// TIA Portal V17 export
// export: Created 2024-09-02T12:49:55.5450562Z, ExportSetting WithDefaults, DisplayName Totally Integrated Automation Portal, DisplayVersion V17, DisplayName TIA Portal Openness, DisplayVersion V17, DisplayName TIA Portal Version Control Interface, DisplayVersion V17, DisplayName STEP 7 Professional, DisplayVersion V17, DisplayName STEP 7 Safety, DisplayVersion V17, DisplayName WinCC Professional, DisplayVersion V17
FUNCTION "SysFC_HMI_Functions" : Void   // FC251, LAD
TITLE = Power supply for function lines / Versorgung Funktionszeilen
{ S7_Optimized_Access := 'TRUE' }
AUTHOR : OlegFuehrus
FAMILY : HMI
NAME : HMI
VERSION : 1.0
// stored: AutoNumber true, IsIECCheckEnabled false, SetENOAutomatically false, UDAEnableTagReadback false
   VAR_INPUT
      "Type" : WString;   // Typ (Setup, PowerUp, Unit, NutRunner, NutRunnerGroup, CycleType, UserDefine) / Type (Setup, PowerUp, Unit, NutRunner, NutRunnerGroup, CycleType, UserDefine)
      Line : Int;   // Zeile (1..348) / Line (1. . 348)
      "Enable Left" : Bool;   // Funktionsfreigabe Links / Functional Approve
      "Enable Right" : Bool;   // Funktionsfreigabe Rechts / Function release right
      "End Pos. Left" : Bool;   // Endlage Links (gelb) / End position Left (yellow)
      "End Pos. Right" : Bool;   // Endlage Rechts (gruen) / End position right (green)
      Position : LReal;   // Positionsanzeige / position display
      "Hide Pos." : Bool;   // Position ausblenden / Hide position
      "Hide Left Arrow" : Bool;   // Pfeil Links ausblenden / Hide left arrow
      "Hide Right Arrow" : Bool;   // Pfeil Rechts ausblenden / Hide left arrow
   END_VAR
   VAR_OUTPUT
      Function_left : Bool;   // Funktionstaste links / Function key left
      Function_right : Bool;   // Funktionstaste rechts / Function key right
      ConfigFault : Bool;   // Configurationsfehler / configuration error
   END_VAR
   VAR_IN_OUT
      LTLL_Config : "LTLL_typeConfig";
      LTLL_Data : "LTLL_typeData";
   END_VAR
   VAR_TEMP
      t_RetVal : Word;
      t_VKE0 : Bool;
      t_VKE1 : Bool;
      t_ConfigFault : Bool;
      t_ConfigFaultNr : Int;
      t_Line : Int;
      t_Line_Uint : UInt;
      t_Btn_Left : Bool;
      t_Btn_Right : Bool;
      t_secure_bit_ok : Bool;
      t_ErrID : Word;
      t_loop : Int;
      t_Pointer : Int;
      t_CmpOK : Bool;
      t_PowerUp : Bool;
   END_VAR
BEGIN

REGION Network 1: VKE0
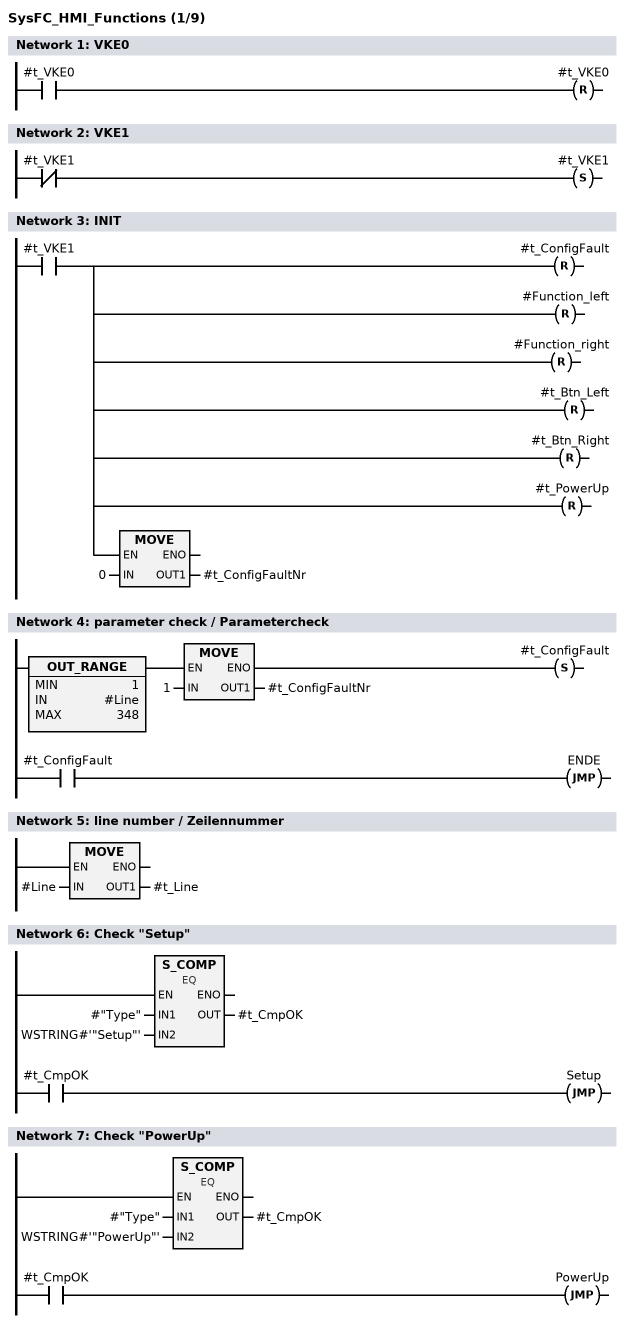
   RUNG wire#powerrail
      Contact( #t_VKE0 )
      R_Coil( #t_VKE0 )
   END_RUNG
   // the same network as SCL:
   IF #t_VKE0 THEN #t_VKE0 := FALSE; END_IF;
END_REGION

REGION Network 2: VKE1
   RUNG wire#powerrail
      I_Contact( #t_VKE1 )
      S_Coil( #t_VKE1 )
   END_RUNG
   // the same network as SCL:
   IF NOT #t_VKE1 THEN #t_VKE1 := TRUE; END_IF;
END_REGION

REGION Network 3: INIT
   RUNG wire#powerrail
      Contact( #t_VKE1 )
      wire#w1
      R_Coil( #t_ConfigFault )
   END_RUNG
   RUNG wire#w1
      R_Coil( #Function_left )
   END_RUNG
   RUNG wire#w1
      R_Coil( #Function_right )
   END_RUNG
   RUNG wire#w1
      R_Coil( #t_Btn_Left )
   END_RUNG
   RUNG wire#w1
      R_Coil( #t_Btn_Right )
   END_RUNG
   RUNG wire#w1
      R_Coil( #t_PowerUp )
   END_RUNG
   RUNG wire#w1
      Move(in := 0, out1 => #t_ConfigFaultNr)
   END_RUNG
   // the same network as SCL:
   IF #t_VKE1 THEN
       #t_ConfigFault := FALSE;
       #Function_left := FALSE;
       #Function_right := FALSE;
       #t_Btn_Left := FALSE;
       #t_Btn_Right := FALSE;
       #t_PowerUp := FALSE;
       #t_ConfigFaultNr := 0;
   END_IF;
END_REGION

REGION Network 4: parameter check / Parametercheck
   IF (#Line < 1) OR (#Line > 348) THEN
       #t_ConfigFaultNr := 1;
       #t_ConfigFault := TRUE;
   END_IF;
   IF #t_ConfigFault THEN GOTO ENDE; END_IF;
END_REGION

REGION Network 5: line number / Zeilennummer
   RUNG wire#powerrail
      Move(in := #Line, out1 => #t_Line)
   END_RUNG
   // the same network as SCL:
   #t_Line := #Line;
END_REGION

REGION Network 6: Check "Setup"
   RUNG wire#powerrail
      { S7_Templates := "[relation := EQ, src_type := WString]" } S_COMP(IN1 := #"Type", IN2 := WSTRING#'"Setup"', OUT => #t_CmpOK)
   END_RUNG
   RUNG wire#powerrail
      Contact( #t_CmpOK )
      JumpCoil( Setup )
   END_RUNG
   // the same network as SCL:
   S_COMP(IN1 := #"Type", IN2 := WSTRING#'"Setup"', OUT => #t_CmpOK);
   IF #t_CmpOK THEN GOTO Setup; END_IF;
END_REGION

REGION Network 7: Check "PowerUp"
   RUNG wire#powerrail
      { S7_Templates := "[relation := EQ, src_type := WString]" } S_COMP(IN1 := #"Type", IN2 := WSTRING#'"PowerUp"', OUT => #t_CmpOK)
   END_RUNG
   RUNG wire#powerrail
      Contact( #t_CmpOK )
      JumpCoil( PowerUp )
   END_RUNG
   // the same network as SCL:
   S_COMP(IN1 := #"Type", IN2 := WSTRING#'"PowerUp"', OUT => #t_CmpOK);
   IF #t_CmpOK THEN GOTO PowerUp; END_IF;
END_REGION

REGION Network 8: Check "Unit"
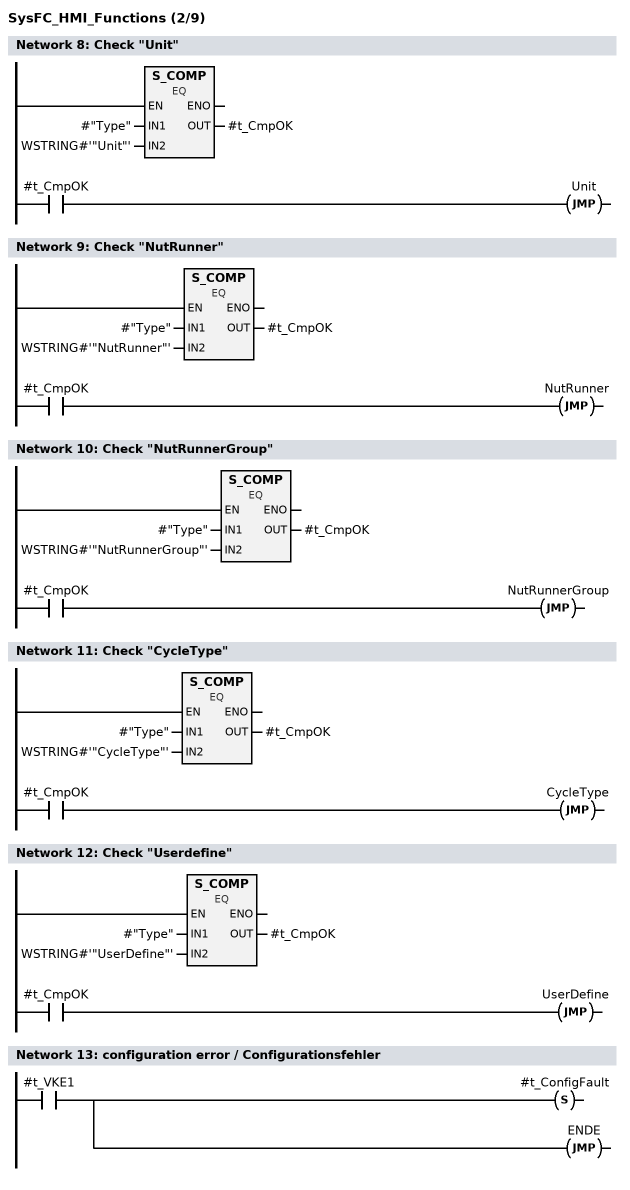
   RUNG wire#powerrail
      { S7_Templates := "[relation := EQ, src_type := WString]" } S_COMP(IN1 := #"Type", IN2 := WSTRING#'"Unit"', OUT => #t_CmpOK)
   END_RUNG
   RUNG wire#powerrail
      Contact( #t_CmpOK )
      JumpCoil( Unit )
   END_RUNG
   // the same network as SCL:
   S_COMP(IN1 := #"Type", IN2 := WSTRING#'"Unit"', OUT => #t_CmpOK);
   IF #t_CmpOK THEN GOTO Unit; END_IF;
END_REGION

REGION Network 9: Check "NutRunner"
   RUNG wire#powerrail
      { S7_Templates := "[relation := EQ, src_type := WString]" } S_COMP(IN1 := #"Type", IN2 := WSTRING#'"NutRunner"', OUT => #t_CmpOK)
   END_RUNG
   RUNG wire#powerrail
      Contact( #t_CmpOK )
      JumpCoil( NutRunner )
   END_RUNG
   // the same network as SCL:
   S_COMP(IN1 := #"Type", IN2 := WSTRING#'"NutRunner"', OUT => #t_CmpOK);
   IF #t_CmpOK THEN GOTO NutRunner; END_IF;
END_REGION

REGION Network 10: Check "NutRunnerGroup"
   RUNG wire#powerrail
      { S7_Templates := "[relation := EQ, src_type := WString]" } S_COMP(IN1 := #"Type", IN2 := WSTRING#'"NutRunnerGroup"', OUT => #t_CmpOK)
   END_RUNG
   RUNG wire#powerrail
      Contact( #t_CmpOK )
      JumpCoil( NutRunnerGroup )
   END_RUNG
   // the same network as SCL:
   S_COMP(IN1 := #"Type", IN2 := WSTRING#'"NutRunnerGroup"', OUT => #t_CmpOK);
   IF #t_CmpOK THEN GOTO NutRunnerGroup; END_IF;
END_REGION

REGION Network 11: Check "CycleType"
   RUNG wire#powerrail
      { S7_Templates := "[relation := EQ, src_type := WString]" } S_COMP(IN1 := #"Type", IN2 := WSTRING#'"CycleType"', OUT => #t_CmpOK)
   END_RUNG
   RUNG wire#powerrail
      Contact( #t_CmpOK )
      JumpCoil( CycleType )
   END_RUNG
   // the same network as SCL:
   S_COMP(IN1 := #"Type", IN2 := WSTRING#'"CycleType"', OUT => #t_CmpOK);
   IF #t_CmpOK THEN GOTO CycleType; END_IF;
END_REGION

REGION Network 12: Check "Userdefine"
   RUNG wire#powerrail
      { S7_Templates := "[relation := EQ, src_type := WString]" } S_COMP(IN1 := #"Type", IN2 := WSTRING#'"UserDefine"', OUT => #t_CmpOK)
   END_RUNG
   RUNG wire#powerrail
      Contact( #t_CmpOK )
      JumpCoil( UserDefine )
   END_RUNG
   // the same network as SCL:
   S_COMP(IN1 := #"Type", IN2 := WSTRING#'"UserDefine"', OUT => #t_CmpOK);
   IF #t_CmpOK THEN GOTO UserDefine; END_IF;
END_REGION

REGION Network 13: configuration error / Configurationsfehler
   RUNG wire#powerrail
      Contact( #t_VKE1 )
      wire#w1
      S_Coil( #t_ConfigFault )
   END_RUNG
   RUNG wire#w1
      JumpCoil( ENDE )
   END_RUNG
   // the same network as SCL:
   IF #t_VKE1 THEN
       #t_ConfigFault := TRUE;
       GOTO ENDE;
   END_IF;
END_REGION

REGION Network 14: Setup
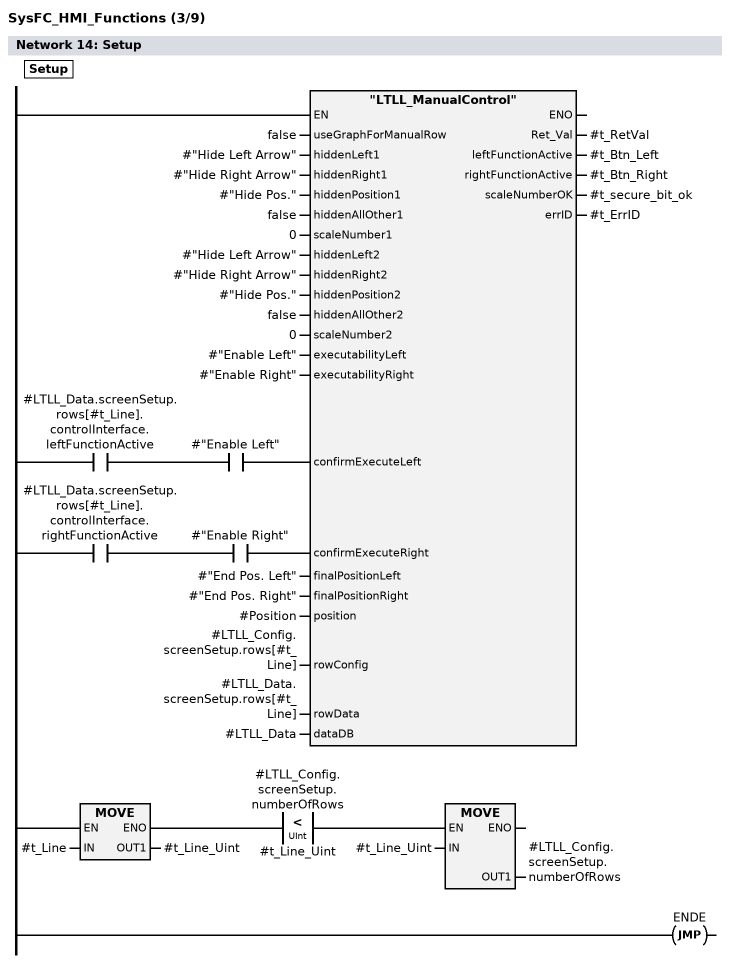
   Label( Setup )
   RUNG wire#powerrail
      "LTLL_ManualControl"(confirmExecuteLeft := wire#w1, confirmExecuteRight := wire#w2, useGraphForManualRow := false, hiddenLeft1 := #"Hide Left Arrow", hiddenRight1 := #"Hide Right Arrow", hiddenPosition1 := #"Hide Pos.", hiddenAllOther1 := false, scaleNumber1 := 0, hiddenLeft2 := #"Hide Left Arrow", hiddenRight2 := #"Hide Right Arrow", hiddenPosition2 := #"Hide Pos.", hiddenAllOther2 := false, scaleNumber2 := 0, executabilityLeft := #"Enable Left", executabilityRight := #"Enable Right", finalPositionLeft := #"End Pos. Left", finalPositionRight := #"End Pos. Right", position := #Position, rowConfig := #LTLL_Config.screenSetup.rows[#t_Line], rowData := #LTLL_Data.screenSetup.rows[#t_Line], dataDB := #LTLL_Data, Ret_Val => #t_RetVal, leftFunctionActive => #t_Btn_Left, rightFunctionActive => #t_Btn_Right, scaleNumberOK => #t_secure_bit_ok, errID => #t_ErrID)
   END_RUNG
   RUNG wire#powerrail
      Contact( #LTLL_Data.screenSetup.rows[#t_Line].controlInterface.leftFunctionActive )
      Contact( #"Enable Left" )
   END_RUNG wire#w1
   RUNG wire#powerrail
      Contact( #LTLL_Data.screenSetup.rows[#t_Line].controlInterface.rightFunctionActive )
      Contact( #"Enable Right" )
   END_RUNG wire#w2
   RUNG wire#powerrail
      Move(in := #t_Line, out1 => #t_Line_Uint)
      { S7_Templates := "SrcType := UInt" } LT_Contact(in1 := #LTLL_Config.screenSetup.numberOfRows, in2 := #t_Line_Uint)
      Move(in := #t_Line_Uint, out1 => #LTLL_Config.screenSetup.numberOfRows)
   END_RUNG
   RUNG wire#powerrail
      JumpCoil( ENDE )
   END_RUNG
   // the same network as SCL:
   Setup:
   #t_RetVal := "LTLL_ManualControl"(useGraphForManualRow := false,
                           hiddenLeft1 := #"Hide Left Arrow",
                           hiddenRight1 := #"Hide Right Arrow",
                           hiddenPosition1 := #"Hide Pos.",
                           hiddenAllOther1 := false,
                           scaleNumber1 := 0,
                           hiddenLeft2 := #"Hide Left Arrow",
                           hiddenRight2 := #"Hide Right Arrow",
                           hiddenPosition2 := #"Hide Pos.",
                           hiddenAllOther2 := false,
                           scaleNumber2 := 0,
                           executabilityLeft := #"Enable Left",
                           executabilityRight := #"Enable Right",
                           confirmExecuteLeft := #LTLL_Data.screenSetup.rows[#t_Line].controlInterface.leftFunctionActive AND #"Enable Left",
                           confirmExecuteRight := #LTLL_Data.screenSetup.rows[#t_Line].controlInterface.rightFunctionActive AND #"Enable Right",
                           finalPositionLeft := #"End Pos. Left",
                           finalPositionRight := #"End Pos. Right",
                           position := #Position,
                           rowConfig := #LTLL_Config.screenSetup.rows[#t_Line],
                           rowData := #LTLL_Data.screenSetup.rows[#t_Line],
                           dataDB := #LTLL_Data,
                           leftFunctionActive => #t_Btn_Left,
                           rightFunctionActive => #t_Btn_Right,
                           scaleNumberOK => #t_secure_bit_ok,
                           errID => #t_ErrID);
   #t_Line_Uint := #t_Line;
   IF #LTLL_Config.screenSetup.numberOfRows < #t_Line_Uint THEN
       #LTLL_Config.screenSetup.numberOfRows := #t_Line_Uint;
   END_IF;
   GOTO ENDE;
END_REGION

REGION Network 15: PowerUp
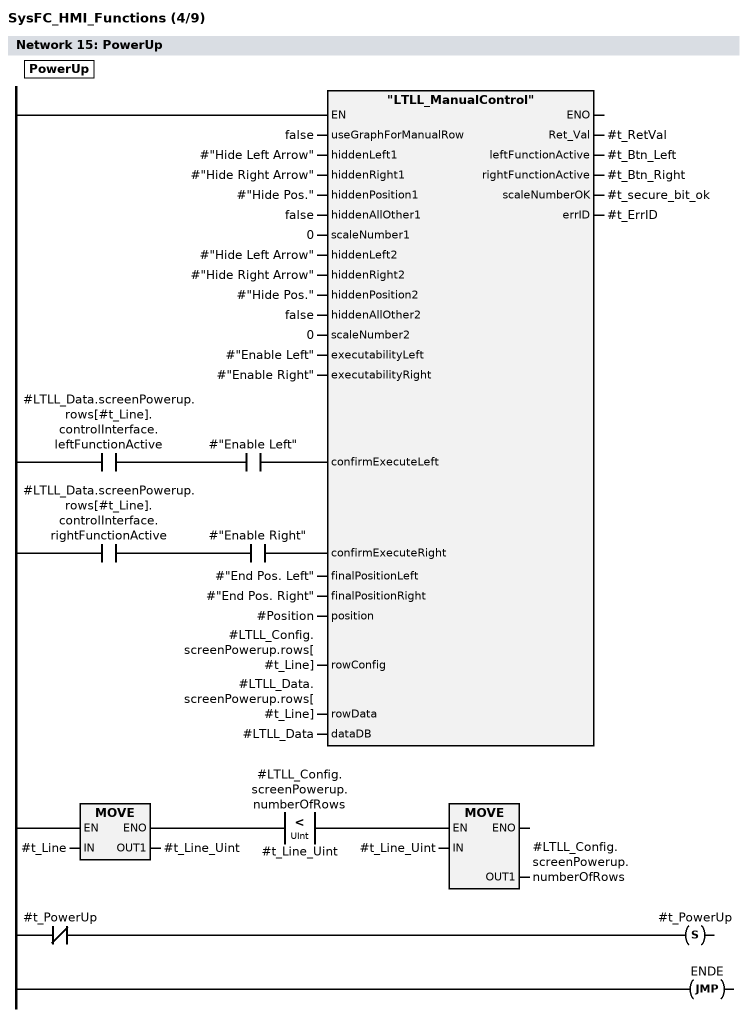
   Label( PowerUp )
   RUNG wire#powerrail
      "LTLL_ManualControl"(confirmExecuteLeft := wire#w1, confirmExecuteRight := wire#w2, useGraphForManualRow := false, hiddenLeft1 := #"Hide Left Arrow", hiddenRight1 := #"Hide Right Arrow", hiddenPosition1 := #"Hide Pos.", hiddenAllOther1 := false, scaleNumber1 := 0, hiddenLeft2 := #"Hide Left Arrow", hiddenRight2 := #"Hide Right Arrow", hiddenPosition2 := #"Hide Pos.", hiddenAllOther2 := false, scaleNumber2 := 0, executabilityLeft := #"Enable Left", executabilityRight := #"Enable Right", finalPositionLeft := #"End Pos. Left", finalPositionRight := #"End Pos. Right", position := #Position, rowConfig := #LTLL_Config.screenPowerup.rows[#t_Line], rowData := #LTLL_Data.screenPowerup.rows[#t_Line], dataDB := #LTLL_Data, Ret_Val => #t_RetVal, leftFunctionActive => #t_Btn_Left, rightFunctionActive => #t_Btn_Right, scaleNumberOK => #t_secure_bit_ok, errID => #t_ErrID)
   END_RUNG
   RUNG wire#powerrail
      Contact( #LTLL_Data.screenPowerup.rows[#t_Line].controlInterface.leftFunctionActive )
      Contact( #"Enable Left" )
   END_RUNG wire#w1
   RUNG wire#powerrail
      Contact( #LTLL_Data.screenPowerup.rows[#t_Line].controlInterface.rightFunctionActive )
      Contact( #"Enable Right" )
   END_RUNG wire#w2
   RUNG wire#powerrail
      Move(in := #t_Line, out1 => #t_Line_Uint)
      { S7_Templates := "SrcType := UInt" } LT_Contact(in1 := #LTLL_Config.screenPowerup.numberOfRows, in2 := #t_Line_Uint)
      Move(in := #t_Line_Uint, out1 => #LTLL_Config.screenPowerup.numberOfRows)
   END_RUNG
   RUNG wire#powerrail
      I_Contact( #t_PowerUp )
      S_Coil( #t_PowerUp )
   END_RUNG
   RUNG wire#powerrail
      JumpCoil( ENDE )
   END_RUNG
   // the same network as SCL:
   PowerUp:
   #t_RetVal := "LTLL_ManualControl"(useGraphForManualRow := false,
                           hiddenLeft1 := #"Hide Left Arrow",
                           hiddenRight1 := #"Hide Right Arrow",
                           hiddenPosition1 := #"Hide Pos.",
                           hiddenAllOther1 := false,
                           scaleNumber1 := 0,
                           hiddenLeft2 := #"Hide Left Arrow",
                           hiddenRight2 := #"Hide Right Arrow",
                           hiddenPosition2 := #"Hide Pos.",
                           hiddenAllOther2 := false,
                           scaleNumber2 := 0,
                           executabilityLeft := #"Enable Left",
                           executabilityRight := #"Enable Right",
                           confirmExecuteLeft := #LTLL_Data.screenPowerup.rows[#t_Line].controlInterface.leftFunctionActive AND #"Enable Left",
                           confirmExecuteRight := #LTLL_Data.screenPowerup.rows[#t_Line].controlInterface.rightFunctionActive AND #"Enable Right",
                           finalPositionLeft := #"End Pos. Left",
                           finalPositionRight := #"End Pos. Right",
                           position := #Position,
                           rowConfig := #LTLL_Config.screenPowerup.rows[#t_Line],
                           rowData := #LTLL_Data.screenPowerup.rows[#t_Line],
                           dataDB := #LTLL_Data,
                           leftFunctionActive => #t_Btn_Left,
                           rightFunctionActive => #t_Btn_Right,
                           scaleNumberOK => #t_secure_bit_ok,
                           errID => #t_ErrID);
   #t_Line_Uint := #t_Line;
   IF #LTLL_Config.screenPowerup.numberOfRows < #t_Line_Uint THEN
       #LTLL_Config.screenPowerup.numberOfRows := #t_Line_Uint;
   END_IF;
   IF NOT #t_PowerUp THEN #t_PowerUp := TRUE; END_IF;
   GOTO ENDE;
END_REGION

REGION Network 16: Unit
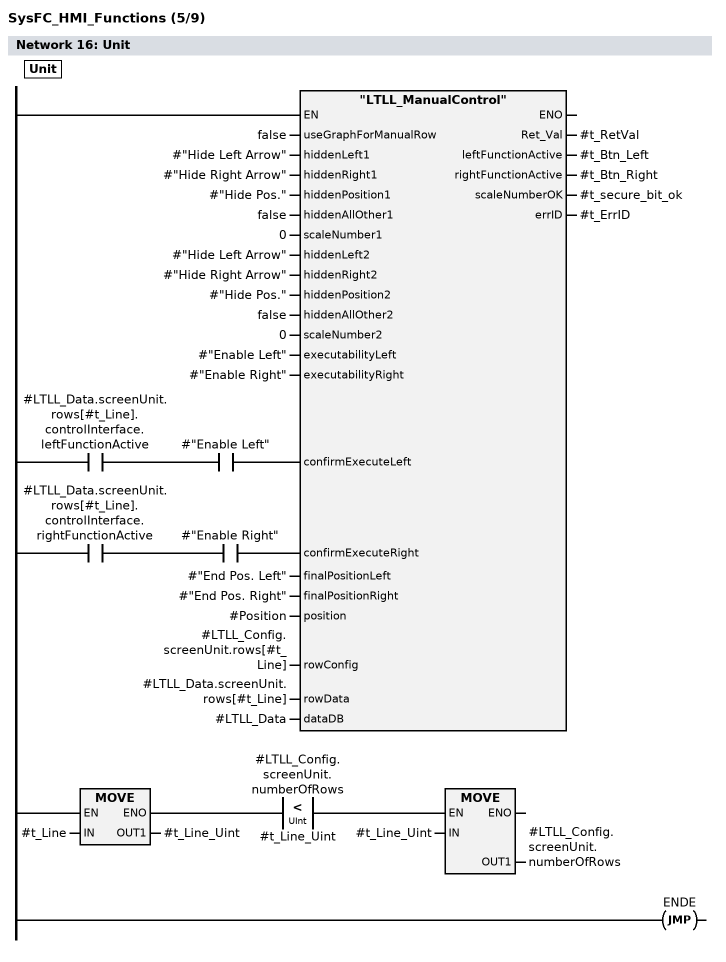
   Label( Unit )
   RUNG wire#powerrail
      "LTLL_ManualControl"(confirmExecuteLeft := wire#w1, confirmExecuteRight := wire#w2, useGraphForManualRow := false, hiddenLeft1 := #"Hide Left Arrow", hiddenRight1 := #"Hide Right Arrow", hiddenPosition1 := #"Hide Pos.", hiddenAllOther1 := false, scaleNumber1 := 0, hiddenLeft2 := #"Hide Left Arrow", hiddenRight2 := #"Hide Right Arrow", hiddenPosition2 := #"Hide Pos.", hiddenAllOther2 := false, scaleNumber2 := 0, executabilityLeft := #"Enable Left", executabilityRight := #"Enable Right", finalPositionLeft := #"End Pos. Left", finalPositionRight := #"End Pos. Right", position := #Position, rowConfig := #LTLL_Config.screenUnit.rows[#t_Line], rowData := #LTLL_Data.screenUnit.rows[#t_Line], dataDB := #LTLL_Data, Ret_Val => #t_RetVal, leftFunctionActive => #t_Btn_Left, rightFunctionActive => #t_Btn_Right, scaleNumberOK => #t_secure_bit_ok, errID => #t_ErrID)
   END_RUNG
   RUNG wire#powerrail
      Contact( #LTLL_Data.screenUnit.rows[#t_Line].controlInterface.leftFunctionActive )
      Contact( #"Enable Left" )
   END_RUNG wire#w1
   RUNG wire#powerrail
      Contact( #LTLL_Data.screenUnit.rows[#t_Line].controlInterface.rightFunctionActive )
      Contact( #"Enable Right" )
   END_RUNG wire#w2
   RUNG wire#powerrail
      Move(in := #t_Line, out1 => #t_Line_Uint)
      { S7_Templates := "SrcType := UInt" } LT_Contact(in1 := #LTLL_Config.screenUnit.numberOfRows, in2 := #t_Line_Uint)
      Move(in := #t_Line_Uint, out1 => #LTLL_Config.screenUnit.numberOfRows)
   END_RUNG
   RUNG wire#powerrail
      JumpCoil( ENDE )
   END_RUNG
   // the same network as SCL:
   Unit:
   #t_RetVal := "LTLL_ManualControl"(useGraphForManualRow := false,
                           hiddenLeft1 := #"Hide Left Arrow",
                           hiddenRight1 := #"Hide Right Arrow",
                           hiddenPosition1 := #"Hide Pos.",
                           hiddenAllOther1 := false,
                           scaleNumber1 := 0,
                           hiddenLeft2 := #"Hide Left Arrow",
                           hiddenRight2 := #"Hide Right Arrow",
                           hiddenPosition2 := #"Hide Pos.",
                           hiddenAllOther2 := false,
                           scaleNumber2 := 0,
                           executabilityLeft := #"Enable Left",
                           executabilityRight := #"Enable Right",
                           confirmExecuteLeft := #LTLL_Data.screenUnit.rows[#t_Line].controlInterface.leftFunctionActive AND #"Enable Left",
                           confirmExecuteRight := #LTLL_Data.screenUnit.rows[#t_Line].controlInterface.rightFunctionActive AND #"Enable Right",
                           finalPositionLeft := #"End Pos. Left",
                           finalPositionRight := #"End Pos. Right",
                           position := #Position,
                           rowConfig := #LTLL_Config.screenUnit.rows[#t_Line],
                           rowData := #LTLL_Data.screenUnit.rows[#t_Line],
                           dataDB := #LTLL_Data,
                           leftFunctionActive => #t_Btn_Left,
                           rightFunctionActive => #t_Btn_Right,
                           scaleNumberOK => #t_secure_bit_ok,
                           errID => #t_ErrID);
   #t_Line_Uint := #t_Line;
   IF #LTLL_Config.screenUnit.numberOfRows < #t_Line_Uint THEN
       #LTLL_Config.screenUnit.numberOfRows := #t_Line_Uint;
   END_IF;
   GOTO ENDE;
END_REGION

REGION Network 17: NutRunner
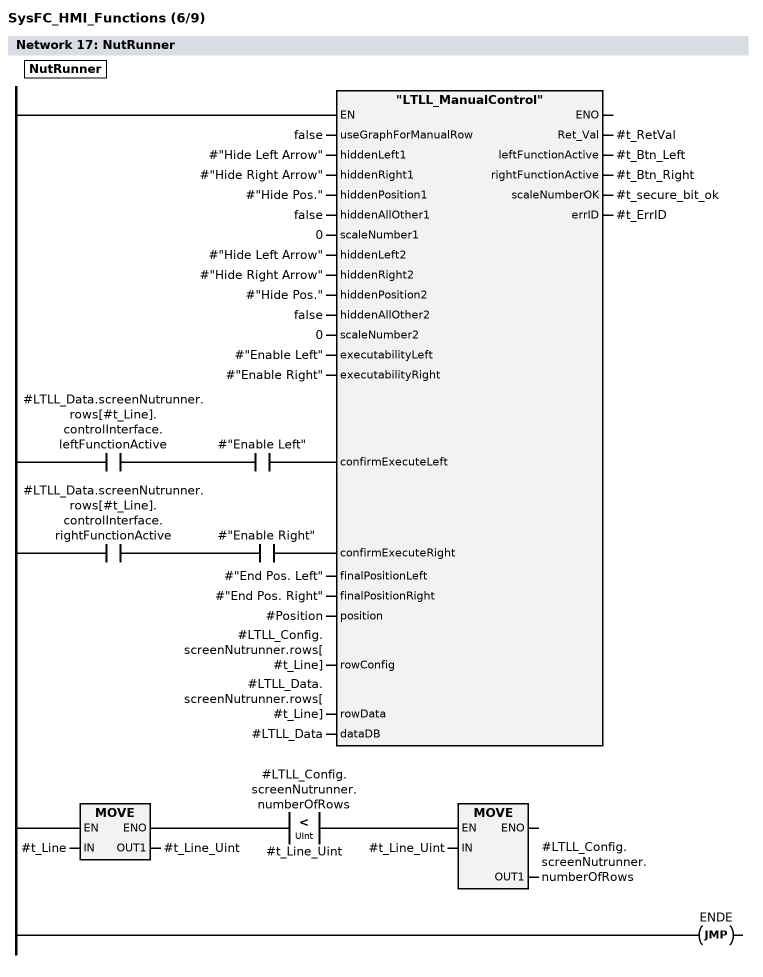
   Label( NutRunner )
   RUNG wire#powerrail
      "LTLL_ManualControl"(confirmExecuteLeft := wire#w1, confirmExecuteRight := wire#w2, useGraphForManualRow := false, hiddenLeft1 := #"Hide Left Arrow", hiddenRight1 := #"Hide Right Arrow", hiddenPosition1 := #"Hide Pos.", hiddenAllOther1 := false, scaleNumber1 := 0, hiddenLeft2 := #"Hide Left Arrow", hiddenRight2 := #"Hide Right Arrow", hiddenPosition2 := #"Hide Pos.", hiddenAllOther2 := false, scaleNumber2 := 0, executabilityLeft := #"Enable Left", executabilityRight := #"Enable Right", finalPositionLeft := #"End Pos. Left", finalPositionRight := #"End Pos. Right", position := #Position, rowConfig := #LTLL_Config.screenNutrunner.rows[#t_Line], rowData := #LTLL_Data.screenNutrunner.rows[#t_Line], dataDB := #LTLL_Data, Ret_Val => #t_RetVal, leftFunctionActive => #t_Btn_Left, rightFunctionActive => #t_Btn_Right, scaleNumberOK => #t_secure_bit_ok, errID => #t_ErrID)
   END_RUNG
   RUNG wire#powerrail
      Contact( #LTLL_Data.screenNutrunner.rows[#t_Line].controlInterface.leftFunctionActive )
      Contact( #"Enable Left" )
   END_RUNG wire#w1
   RUNG wire#powerrail
      Contact( #LTLL_Data.screenNutrunner.rows[#t_Line].controlInterface.rightFunctionActive )
      Contact( #"Enable Right" )
   END_RUNG wire#w2
   RUNG wire#powerrail
      Move(in := #t_Line, out1 => #t_Line_Uint)
      { S7_Templates := "SrcType := UInt" } LT_Contact(in1 := #LTLL_Config.screenNutrunner.numberOfRows, in2 := #t_Line_Uint)
      Move(in := #t_Line_Uint, out1 => #LTLL_Config.screenNutrunner.numberOfRows)
   END_RUNG
   RUNG wire#powerrail
      JumpCoil( ENDE )
   END_RUNG
   // the same network as SCL:
   NutRunner:
   #t_RetVal := "LTLL_ManualControl"(useGraphForManualRow := false,
                           hiddenLeft1 := #"Hide Left Arrow",
                           hiddenRight1 := #"Hide Right Arrow",
                           hiddenPosition1 := #"Hide Pos.",
                           hiddenAllOther1 := false,
                           scaleNumber1 := 0,
                           hiddenLeft2 := #"Hide Left Arrow",
                           hiddenRight2 := #"Hide Right Arrow",
                           hiddenPosition2 := #"Hide Pos.",
                           hiddenAllOther2 := false,
                           scaleNumber2 := 0,
                           executabilityLeft := #"Enable Left",
                           executabilityRight := #"Enable Right",
                           confirmExecuteLeft := #LTLL_Data.screenNutrunner.rows[#t_Line].controlInterface.leftFunctionActive AND #"Enable Left",
                           confirmExecuteRight := #LTLL_Data.screenNutrunner.rows[#t_Line].controlInterface.rightFunctionActive AND #"Enable Right",
                           finalPositionLeft := #"End Pos. Left",
                           finalPositionRight := #"End Pos. Right",
                           position := #Position,
                           rowConfig := #LTLL_Config.screenNutrunner.rows[#t_Line],
                           rowData := #LTLL_Data.screenNutrunner.rows[#t_Line],
                           dataDB := #LTLL_Data,
                           leftFunctionActive => #t_Btn_Left,
                           rightFunctionActive => #t_Btn_Right,
                           scaleNumberOK => #t_secure_bit_ok,
                           errID => #t_ErrID);
   #t_Line_Uint := #t_Line;
   IF #LTLL_Config.screenNutrunner.numberOfRows < #t_Line_Uint THEN
       #LTLL_Config.screenNutrunner.numberOfRows := #t_Line_Uint;
   END_IF;
   GOTO ENDE;
END_REGION

REGION Network 18: NutRunnerGroup
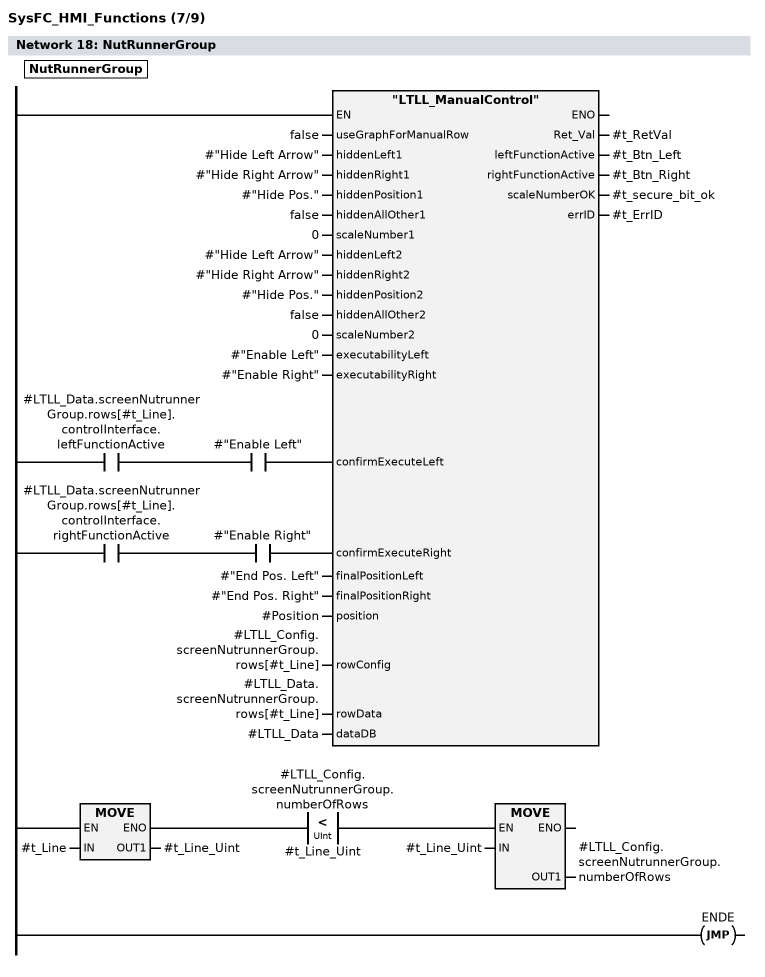
   Label( NutRunnerGroup )
   RUNG wire#powerrail
      "LTLL_ManualControl"(confirmExecuteLeft := wire#w1, confirmExecuteRight := wire#w2, useGraphForManualRow := false, hiddenLeft1 := #"Hide Left Arrow", hiddenRight1 := #"Hide Right Arrow", hiddenPosition1 := #"Hide Pos.", hiddenAllOther1 := false, scaleNumber1 := 0, hiddenLeft2 := #"Hide Left Arrow", hiddenRight2 := #"Hide Right Arrow", hiddenPosition2 := #"Hide Pos.", hiddenAllOther2 := false, scaleNumber2 := 0, executabilityLeft := #"Enable Left", executabilityRight := #"Enable Right", finalPositionLeft := #"End Pos. Left", finalPositionRight := #"End Pos. Right", position := #Position, rowConfig := #LTLL_Config.screenNutrunnerGroup.rows[#t_Line], rowData := #LTLL_Data.screenNutrunnerGroup.rows[#t_Line], dataDB := #LTLL_Data, Ret_Val => #t_RetVal, leftFunctionActive => #t_Btn_Left, rightFunctionActive => #t_Btn_Right, scaleNumberOK => #t_secure_bit_ok, errID => #t_ErrID)
   END_RUNG
   RUNG wire#powerrail
      Contact( #LTLL_Data.screenNutrunnerGroup.rows[#t_Line].controlInterface.leftFunctionActive )
      Contact( #"Enable Left" )
   END_RUNG wire#w1
   RUNG wire#powerrail
      Contact( #LTLL_Data.screenNutrunnerGroup.rows[#t_Line].controlInterface.rightFunctionActive )
      Contact( #"Enable Right" )
   END_RUNG wire#w2
   RUNG wire#powerrail
      Move(in := #t_Line, out1 => #t_Line_Uint)
      { S7_Templates := "SrcType := UInt" } LT_Contact(in1 := #LTLL_Config.screenNutrunnerGroup.numberOfRows, in2 := #t_Line_Uint)
      Move(in := #t_Line_Uint, out1 => #LTLL_Config.screenNutrunnerGroup.numberOfRows)
   END_RUNG
   RUNG wire#powerrail
      JumpCoil( ENDE )
   END_RUNG
   // the same network as SCL:
   NutRunnerGroup:
   #t_RetVal := "LTLL_ManualControl"(useGraphForManualRow := false,
                           hiddenLeft1 := #"Hide Left Arrow",
                           hiddenRight1 := #"Hide Right Arrow",
                           hiddenPosition1 := #"Hide Pos.",
                           hiddenAllOther1 := false,
                           scaleNumber1 := 0,
                           hiddenLeft2 := #"Hide Left Arrow",
                           hiddenRight2 := #"Hide Right Arrow",
                           hiddenPosition2 := #"Hide Pos.",
                           hiddenAllOther2 := false,
                           scaleNumber2 := 0,
                           executabilityLeft := #"Enable Left",
                           executabilityRight := #"Enable Right",
                           confirmExecuteLeft := #LTLL_Data.screenNutrunnerGroup.rows[#t_Line].controlInterface.leftFunctionActive AND #"Enable Left",
                           confirmExecuteRight := #LTLL_Data.screenNutrunnerGroup.rows[#t_Line].controlInterface.rightFunctionActive AND #"Enable Right",
                           finalPositionLeft := #"End Pos. Left",
                           finalPositionRight := #"End Pos. Right",
                           position := #Position,
                           rowConfig := #LTLL_Config.screenNutrunnerGroup.rows[#t_Line],
                           rowData := #LTLL_Data.screenNutrunnerGroup.rows[#t_Line],
                           dataDB := #LTLL_Data,
                           leftFunctionActive => #t_Btn_Left,
                           rightFunctionActive => #t_Btn_Right,
                           scaleNumberOK => #t_secure_bit_ok,
                           errID => #t_ErrID);
   #t_Line_Uint := #t_Line;
   IF #LTLL_Config.screenNutrunnerGroup.numberOfRows < #t_Line_Uint THEN
       #LTLL_Config.screenNutrunnerGroup.numberOfRows := #t_Line_Uint;
   END_IF;
   GOTO ENDE;
END_REGION

REGION Network 19: CycleType
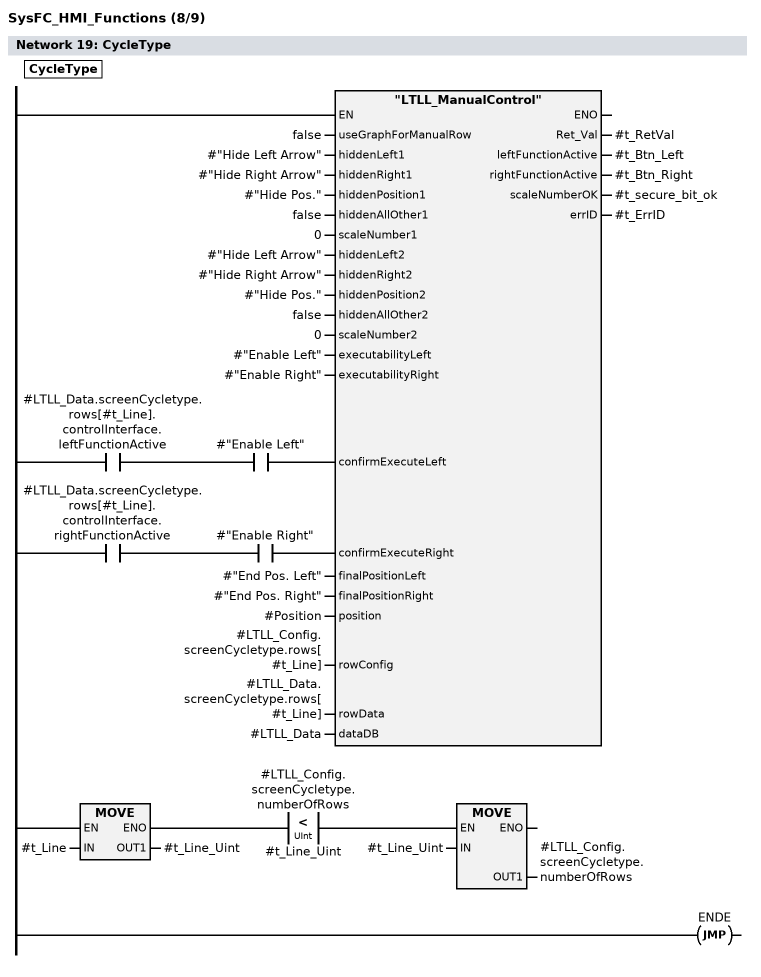
   Label( CycleType )
   RUNG wire#powerrail
      "LTLL_ManualControl"(confirmExecuteLeft := wire#w1, confirmExecuteRight := wire#w2, useGraphForManualRow := false, hiddenLeft1 := #"Hide Left Arrow", hiddenRight1 := #"Hide Right Arrow", hiddenPosition1 := #"Hide Pos.", hiddenAllOther1 := false, scaleNumber1 := 0, hiddenLeft2 := #"Hide Left Arrow", hiddenRight2 := #"Hide Right Arrow", hiddenPosition2 := #"Hide Pos.", hiddenAllOther2 := false, scaleNumber2 := 0, executabilityLeft := #"Enable Left", executabilityRight := #"Enable Right", finalPositionLeft := #"End Pos. Left", finalPositionRight := #"End Pos. Right", position := #Position, rowConfig := #LTLL_Config.screenCycletype.rows[#t_Line], rowData := #LTLL_Data.screenCycletype.rows[#t_Line], dataDB := #LTLL_Data, Ret_Val => #t_RetVal, leftFunctionActive => #t_Btn_Left, rightFunctionActive => #t_Btn_Right, scaleNumberOK => #t_secure_bit_ok, errID => #t_ErrID)
   END_RUNG
   RUNG wire#powerrail
      Contact( #LTLL_Data.screenCycletype.rows[#t_Line].controlInterface.leftFunctionActive )
      Contact( #"Enable Left" )
   END_RUNG wire#w1
   RUNG wire#powerrail
      Contact( #LTLL_Data.screenCycletype.rows[#t_Line].controlInterface.rightFunctionActive )
      Contact( #"Enable Right" )
   END_RUNG wire#w2
   RUNG wire#powerrail
      Move(in := #t_Line, out1 => #t_Line_Uint)
      { S7_Templates := "SrcType := UInt" } LT_Contact(in1 := #LTLL_Config.screenCycletype.numberOfRows, in2 := #t_Line_Uint)
      Move(in := #t_Line_Uint, out1 => #LTLL_Config.screenCycletype.numberOfRows)
   END_RUNG
   RUNG wire#powerrail
      JumpCoil( ENDE )
   END_RUNG
   // the same network as SCL:
   CycleType:
   #t_RetVal := "LTLL_ManualControl"(useGraphForManualRow := false,
                           hiddenLeft1 := #"Hide Left Arrow",
                           hiddenRight1 := #"Hide Right Arrow",
                           hiddenPosition1 := #"Hide Pos.",
                           hiddenAllOther1 := false,
                           scaleNumber1 := 0,
                           hiddenLeft2 := #"Hide Left Arrow",
                           hiddenRight2 := #"Hide Right Arrow",
                           hiddenPosition2 := #"Hide Pos.",
                           hiddenAllOther2 := false,
                           scaleNumber2 := 0,
                           executabilityLeft := #"Enable Left",
                           executabilityRight := #"Enable Right",
                           confirmExecuteLeft := #LTLL_Data.screenCycletype.rows[#t_Line].controlInterface.leftFunctionActive AND #"Enable Left",
                           confirmExecuteRight := #LTLL_Data.screenCycletype.rows[#t_Line].controlInterface.rightFunctionActive AND #"Enable Right",
                           finalPositionLeft := #"End Pos. Left",
                           finalPositionRight := #"End Pos. Right",
                           position := #Position,
                           rowConfig := #LTLL_Config.screenCycletype.rows[#t_Line],
                           rowData := #LTLL_Data.screenCycletype.rows[#t_Line],
                           dataDB := #LTLL_Data,
                           leftFunctionActive => #t_Btn_Left,
                           rightFunctionActive => #t_Btn_Right,
                           scaleNumberOK => #t_secure_bit_ok,
                           errID => #t_ErrID);
   #t_Line_Uint := #t_Line;
   IF #LTLL_Config.screenCycletype.numberOfRows < #t_Line_Uint THEN
       #LTLL_Config.screenCycletype.numberOfRows := #t_Line_Uint;
   END_IF;
   GOTO ENDE;
END_REGION

REGION Network 20: UserDefine
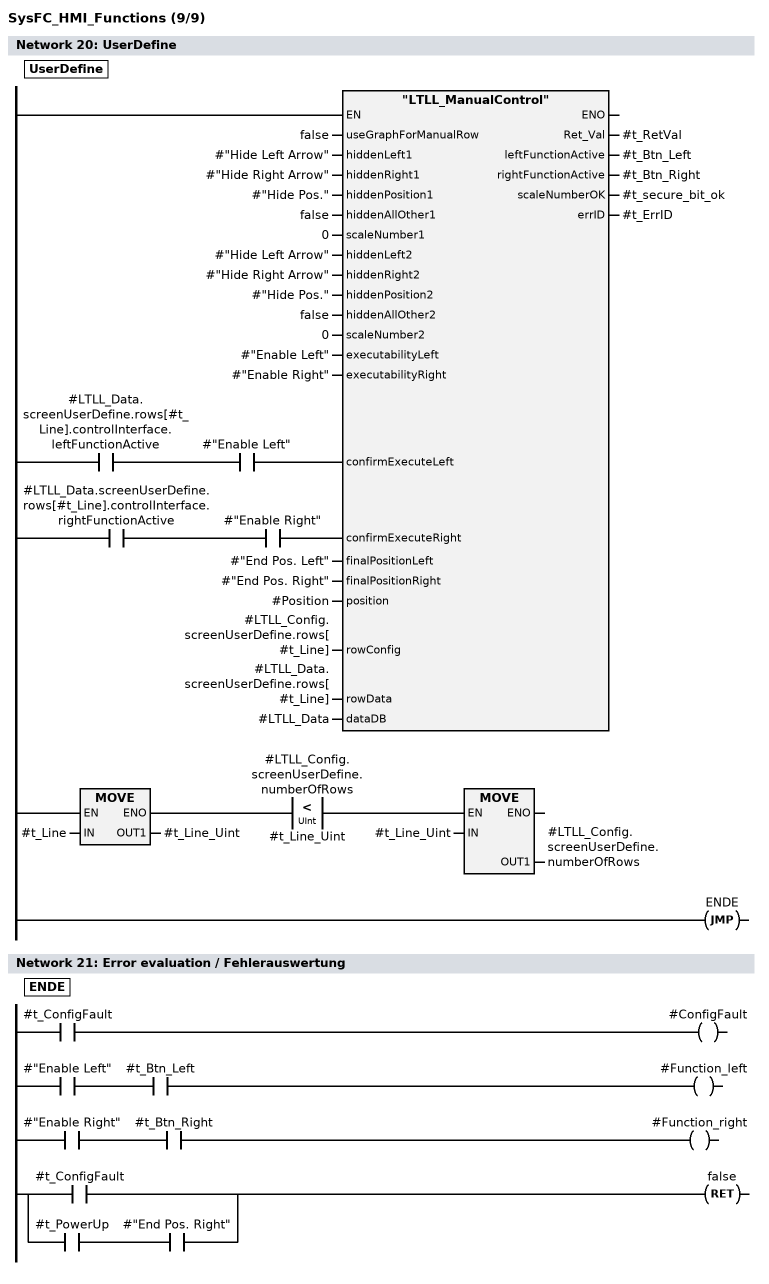
   Label( UserDefine )
   RUNG wire#powerrail
      "LTLL_ManualControl"(confirmExecuteLeft := wire#w1, confirmExecuteRight := wire#w2, useGraphForManualRow := false, hiddenLeft1 := #"Hide Left Arrow", hiddenRight1 := #"Hide Right Arrow", hiddenPosition1 := #"Hide Pos.", hiddenAllOther1 := false, scaleNumber1 := 0, hiddenLeft2 := #"Hide Left Arrow", hiddenRight2 := #"Hide Right Arrow", hiddenPosition2 := #"Hide Pos.", hiddenAllOther2 := false, scaleNumber2 := 0, executabilityLeft := #"Enable Left", executabilityRight := #"Enable Right", finalPositionLeft := #"End Pos. Left", finalPositionRight := #"End Pos. Right", position := #Position, rowConfig := #LTLL_Config.screenUserDefine.rows[#t_Line], rowData := #LTLL_Data.screenUserDefine.rows[#t_Line], dataDB := #LTLL_Data, Ret_Val => #t_RetVal, leftFunctionActive => #t_Btn_Left, rightFunctionActive => #t_Btn_Right, scaleNumberOK => #t_secure_bit_ok, errID => #t_ErrID)
   END_RUNG
   RUNG wire#powerrail
      Contact( #LTLL_Data.screenUserDefine.rows[#t_Line].controlInterface.leftFunctionActive )
      Contact( #"Enable Left" )
   END_RUNG wire#w1
   RUNG wire#powerrail
      Contact( #LTLL_Data.screenUserDefine.rows[#t_Line].controlInterface.rightFunctionActive )
      Contact( #"Enable Right" )
   END_RUNG wire#w2
   RUNG wire#powerrail
      Move(in := #t_Line, out1 => #t_Line_Uint)
      { S7_Templates := "SrcType := UInt" } LT_Contact(in1 := #LTLL_Config.screenUserDefine.numberOfRows, in2 := #t_Line_Uint)
      Move(in := #t_Line_Uint, out1 => #LTLL_Config.screenUserDefine.numberOfRows)
   END_RUNG
   RUNG wire#powerrail
      JumpCoil( ENDE )
   END_RUNG
   // the same network as SCL:
   UserDefine:
   #t_RetVal := "LTLL_ManualControl"(useGraphForManualRow := false,
                           hiddenLeft1 := #"Hide Left Arrow",
                           hiddenRight1 := #"Hide Right Arrow",
                           hiddenPosition1 := #"Hide Pos.",
                           hiddenAllOther1 := false,
                           scaleNumber1 := 0,
                           hiddenLeft2 := #"Hide Left Arrow",
                           hiddenRight2 := #"Hide Right Arrow",
                           hiddenPosition2 := #"Hide Pos.",
                           hiddenAllOther2 := false,
                           scaleNumber2 := 0,
                           executabilityLeft := #"Enable Left",
                           executabilityRight := #"Enable Right",
                           confirmExecuteLeft := #LTLL_Data.screenUserDefine.rows[#t_Line].controlInterface.leftFunctionActive AND #"Enable Left",
                           confirmExecuteRight := #LTLL_Data.screenUserDefine.rows[#t_Line].controlInterface.rightFunctionActive AND #"Enable Right",
                           finalPositionLeft := #"End Pos. Left",
                           finalPositionRight := #"End Pos. Right",
                           position := #Position,
                           rowConfig := #LTLL_Config.screenUserDefine.rows[#t_Line],
                           rowData := #LTLL_Data.screenUserDefine.rows[#t_Line],
                           dataDB := #LTLL_Data,
                           leftFunctionActive => #t_Btn_Left,
                           rightFunctionActive => #t_Btn_Right,
                           scaleNumberOK => #t_secure_bit_ok,
                           errID => #t_ErrID);
   #t_Line_Uint := #t_Line;
   IF #LTLL_Config.screenUserDefine.numberOfRows < #t_Line_Uint THEN
       #LTLL_Config.screenUserDefine.numberOfRows := #t_Line_Uint;
   END_IF;
   GOTO ENDE;
END_REGION

REGION Network 21: Error evaluation / Fehlerauswertung
   ENDE:
   #ConfigFault := #t_ConfigFault;
   #Function_left := #"Enable Left" AND #t_Btn_Left;
   #Function_right := #"Enable Right" AND #t_Btn_Right;
   IF #t_ConfigFault OR (#t_PowerUp AND #"End Pos. Right") THEN
       ENO := false;
       RETURN;
   END_IF;
END_REGION
END_FUNCTION
